(* CODESYS project IODev.library
   Company: ESO
   Description: Local Device Control - LDC IODevLibrary based on State Machine
   Version: 1.1.1.0
   Placeholder: ESO LDC IODev Library
   Author: Dan Popovic
   Title: ESO LDC IODev Library

Project tree, tasks and I/O mapping:
  libraries: Tc2_Standard, * (Beckhoff Automation GmbH); Tc2_System, * (Beckhoff Automation GmbH); Tc3_EventLogger, * (Beckhoff Automation GmbH); Tc3_Module, * (Beckhoff Automation GmbH); VisuSymbols, 3.5.10.0 (System)
  config/
    Device1_EtherCAT_SPLC014.xti
    Mappings_HW_SPLC014.xml
    Mappings_SIM.xml
  00000000-0000-0000-0000-000000000000|config\Device1_EtherCAT_SPLC014.xti
  00000000-0000-0000-0000-000000000000|config\Mappings_HW_SPLC014.xml
  00000000-0000-0000-0000-000000000000|config\Mappings_SIM.xml
  doc/
  DUTs/
    Enumerated/
      data type E_IODEV_COMMAND
      data type E_IODEV_CONVERSION
      data type E_IODEV_ERROR
      data type E_IODEV_EVENT
      data type E_IODEV_RPC_ERROR
      data type E_IODEV_STATE
      data type E_IODEV_STATUS
      data type E_IODEV_SUBSTATE
    Structures/
      data type T_IODEV_CFG
      data type T_IODEV_CTRL
      data type T_IODEV_INFO
      data type T_IODEV_STAT
  GVLs/
  lib/
  POUs/
    Channels/
      function block FB_IODEV_CH_ANALOG [ST]
      function block FB_IODEV_CH_ANLG_IN [ST]: M_Compute, M_Configure, M_Reset
      function block FB_IODEV_CH_ANLG_OUT [ST]: M_Compute, M_Configure, M_Reset
      function block FB_IODEV_CH_DIG_IN [ST]: M_Compute, M_Configure, M_Reset
      function block FB_IODEV_CH_DIG_OUT [ST]: M_Compute, M_Configure, M_Reset
      function block FB_IODEV_CH_DIGITAL [ST]
      function block FB_IODEV_CH_REAL [ST]
      function block FB_IODEV_CH_REAL_IN [ST]: M_Compute, M_Configure, M_Reset
      function block FB_IODEV_CHANNEL [ST]: M_Compute, M_Reset
    Examples/
      function block FB_IODEV_2_4_2_2_USER_CONFIG [ST]: M_UserConfigure
      function block FB_SENS_2_4A_2R_USER_CONFIG [ST]: M_UserConfigure
      function block FB_SENS_8_4 [ST]
      function block FB_SENS_8_4_USER_CONFIG [ST]: M_UserConfigure
      data type T_IODEV_CTRL_2_2
      data type T_IODEV_STAT_2_4
      data type T_IODEV_STAT_2_4A_2R
      data type T_IODEV_STAT_8_4
    Simulation/
      function block FB_SIM_SIGNAL_ANALOG [ST]
      function block FB_SIM_SIGNAL_DIGITAL [ST]
      function block FB_SIM_SIGNAL_REAL [ST]
    function block FB_IODEV_BASE [ST]: ActionDisableExecute, ActionEnableExecute, ActionErrExecute, ActionInitExecute, ActionResetExecute, ActionSetExecute, ActionStopExecute, ActionUnexpExecute, ActivityMonitoring, CheckForEvents, M_Configure, M_GetRpcErrorText, M_LogEventDebug, M_LogEventError, M_LogEventGeneral, M_ReadSensors, M_ResetConfig, M_ResetOutputs, M_SetOutputs, M_SetRpcStatus, M_UserConfigure, ProcessEvents, RPC_Disable, RPC_Enable, RPC_Init, RPC_Reset, RPC_SetDebug, RPC_SetLog, RPC_SetOutputs, RPC_Stop, SetAction, SetEvent, SetLastCommand, SetState, SetStatus
    program MAIN [ST]
  Version/
    global variables Global_Version
  VISUs/
    Templates/
      visualisation GUI_TEMPLATE_IODEV
    visualisation GUI_IODev001
    visualisation GUI_IODev002
  text list GlobalTextList
*)

// DUTs/Enumerated/E_IODEV_COMMAND
{attribute 'qualified_only'}
{attribute 'strict'}
TYPE E_IODEV_COMMAND :
(
	NONE	:= 0,
	
	RESET,
	INIT,
	STOP,
	ENABLE,
	DISABLE,
	SET_OUTPUTS
	
);
END_TYPE

// DUTs/Enumerated/E_IODEV_CONVERSION
TYPE E_IODEV_CONVERSION :
(
	CONVERSION_IODEV_NONE	:= 0,
	
	// Digital signals
	CONVERSION_IODEV_DIGITAL,
	// Analog signals
	CONVERSION_IODEV_LINEAR,
	CONVERSION_IODEV_QUADRATIC,
	CONVERSION_IODEV_EXP,
	CONVERSION_IODEV_EXP10
	
);
END_TYPE

// DUTs/Enumerated/E_IODEV_ERROR
{attribute 'qualified_only'}
{attribute 'strict'}
TYPE E_IODEV_ERROR :
(
	OK					:= 0,
	HW_NOT_OP			:= 1,			
	WRONG_CMD			:= 2,			
	INIT_FAILURE		:= 3,		

	NOT_INITIALISED		:= 90,
	ZERO_POINTER		:= 100	// Simulator error
);
END_TYPE

// DUTs/Enumerated/E_IODEV_EVENT
{attribute 'qualified_only'}
{attribute 'strict'}
TYPE E_IODEV_EVENT :
(
	NONE	:= 0,
	
	(* events corresponding to commands *)
	RESET,
	INIT,
	STOP,
	ENABLE,
	DISABLE,
	SET,
	
	(* 
		Events corresponding to internal events 
	*)
	INITDONE,
	
	
	(* events mapped to HW signals *)
	HWOK,
	ERRHW,
	ERRINIT
	
);
END_TYPE

// DUTs/Enumerated/E_IODEV_RPC_ERROR
{attribute 'qualified_only'}
{attribute 'strict'}
TYPE E_IODEV_RPC_ERROR :
(
	OK						:= 0,
	NOT_OP					:= -1,			
	NOT_NOTOP_READY			:= -2,			
	NOT_NOTOP_NOTREADY		:= -3,			
	LOCAL					:= -4			
);
END_TYPE

// DUTs/Enumerated/E_IODEV_STATE
{attribute 'qualified_only'}
{attribute 'strict'}
TYPE E_IODEV_STATE :
(
	NONE	:= 0,
	NOTOP,
	OP
);
END_TYPE

// DUTs/Enumerated/E_IODEV_STATUS
{attribute 'qualified_only'}
{attribute 'strict'}
TYPE E_IODEV_STATUS :
(
	OK		:= 0,
	ERROR
);
END_TYPE

// DUTs/Enumerated/E_IODEV_SUBSTATE
// Substates MUST match definitions in the WS driver that can be found in
// ICS/ifw/fcf/devmgr/devices/src/include/devmgr/devices/sensorConfig.hpp
// Never change them without consulting the Instrumentation SW team.
{attribute 'qualified_only'}
{attribute 'strict'}
TYPE E_IODEV_SUBSTATE :
(
	NONE			:= 0,
	
	NOTOP_NOTREADY	:= 100,
	NOTOP_READY		:= 101,
	NOTOP_ERROR		:= 199,
	
	OP_MONITORING	:= 200,
	OP_ERROR		:= 299
);
END_TYPE

// DUTs/Structures/T_IODEV_CFG
TYPE T_IODEV_CFG :
STRUCT
	sName:				STRING	:= 'IODev';	// Instance name
	bAutoOp:			BOOL 	:= FALSE;	// If TRUE, go automatically to OPERATIONAL state
	bUserConfig:		BOOL 	:= TRUE;	// If true, configuration in M_Configure() is used.
	
	nNum_DI:			INT		:= 0; 		// Number of digital INPUT signals
	nNum_AI:			INT		:= 0; 		// Number of analog INPUT signals of type INT
	nNum_RI:			INT		:= 0; 		// Number of analog INPUT signals of type REAL
	nNum_DisI:			INT		:= 0; 		// Number of discrete INPUT signals
	nNum_TI:			INT		:= 0; 		// Number of text INPUT signals
	
	nNum_DO:			INT		:= 0; 		// Number of digital OUTPUT signals
	nNum_AO:			INT		:= 0; 		// Number of analog OUTPUT signals of type INT
	nNum_DisO:			INT		:= 0; 		// Number of discrete OUTPUT signals
	nNum_TO:			INT		:= 0; 		// Number of text OUTPUT signals
	
	// Logging
	bLogExtTime:		BOOL 	:= FALSE;		// If TRUE, use external time in event logs. Default FALSE.
	bDebug:				BOOL 	:= FALSE;		// If TRUE, show event logs of Debug type. Default FALSE.
	bLog:				BOOL 	:= TRUE;		// If TRUE, log events. Default TRUE.
	
END_STRUCT
END_TYPE

// DUTs/Structures/T_IODEV_CTRL
TYPE T_IODEV_CTRL :
STRUCT
	nCommand:	E_IODEV_COMMAND	:= E_IODEV_COMMAND.NONE; (* See E_IODEV_COMMAND *)
	bExecute:	BOOL;
	
END_STRUCT
END_TYPE

// DUTs/Structures/T_IODEV_INFO
TYPE T_IODEV_INFO :
STRUCT
(*
Driver Information 

Change Log:
	0.1	2017-09-07	- First version - dummy implementation.
	0.2	2017-09-11	- Implemented digital/analog IN/OUT.
	0.3	2017-09-14	- Implemented digital/analog IN/OUT as FBs with methods.
					- Removed unused structures.
	0.6.0.0			- Restructure with pointers to channel arrays.
					- Removed input vars for number of channels. Defined in each derived FB.
					- Addition of FB_IODEV_SENS_8_4.
					- Addition of customised FB's.
	0.7.0.0			- Addition of stat.sLibVersion
	0.8.0.0			- RPC calls return INT.
					- Addition of E_IODEV_RPC_ERROR.
	0.8.0.1			- Addition of library category ESO/ELT.
	0.8.0.2			- Removed input parameters from OPC UA.
	0.9.0.0			- Renaming States STANDBY->NOTOP & FAILURE->ERROR.
	1.0.0.0			- WARNING: Requires TwinCAT 3.1 build 4022.20 or higher.
					- Projects need Tc3_EventLogger library included in References.
					- Addition of Methods for Event Logs.
					- Addition of cfg.bLog flag for enable/disable of logging.
					- Addition of RPC_SetDebug() and RPC_SetLog().
					- RPC calls not allowed in Local mode.
	1.0.0.1			- Compiled wit TwinCAT 3.1 build 4022.27.
					- Renamed TC_EVENTS.OpsEventClass to TC_EVENTS.IODevOpsEventClass.
					- Solved problem of 'growing' libraries by setting Property/Advanced/BuildAction to None for IODev.library and pdf files in dir config.
	1.0.0.2			- Pinned ST_IODevOpsEventClass under External Types.
	1.0.0.3			- Renumbered enumerations in E_IODEV_SUBSTATE to match WS.
	1.1.0.0			- Moved user defined structures under ctrl and stat.
					- Strict enumerated types.
					- Used RefCtrl and RefStat in BASE FB.
*)
	sDate:			STRING(32)	:= '2019-04-24';
	sDescription:	STRING(80) 	:= 'State Machine based IODev controller';
	sName:			STRING(64)	:= 'FB_IODEV';
	sPlatform:		STRING(32)	:= 'CoDeSys';
	sSynopsis:		STRING(64)	:= 'State Machine based IODev controller';
	nVersionMajor:	DINT		:= 1;
	nVersionMinor:	DINT		:= 1;
END_STRUCT
END_TYPE

// DUTs/Structures/T_IODEV_STAT
TYPE T_IODEV_STAT :
STRUCT
	bLocal:			BOOL	:= FALSE;						(* Device operated from PLC GUI *)

	nState:			E_IODEV_STATE	:= E_IODEV_STATE.NOTOP;				// State
	nSubstate:		E_IODEV_SUBSTATE:= E_IODEV_SUBSTATE.NOTOP_NOTREADY;	// Substate

	nErrorCode: 	E_IODEV_ERROR 	:= E_IODEV_ERROR.OK;		(* Error code *)
	nLastCommand:	E_IODEV_COMMAND	:= E_IODEV_COMMAND.NONE;	(* Last command sent to the device *)
	nRpcErrorCode: 	E_IODEV_RPC_ERROR 	:= E_IODEV_RPC_ERROR.OK;(* RPC Error code *)
	nStatus: 		E_IODEV_STATUS	:= E_IODEV_STATUS.OK; 		(* Device status *)

	sState:			STRING	:= 'NOT OP';					(* State textual description *)
	sSubstate:		STRING	:= 'NOT READY';					(* Substate textual description *)
	sErrorText: 	STRING 	:= 'OK'; 						(* Error text *)
	sRPCErrorText: 	STRING 	:= 'OK'; 						(* RPC Error text *)
	sStatus: 		STRING 	:= 'OK'; 						(* Status in textual form, e.g. 'OFF' *)
	sLastCommand:	STRING	:= 'NONE';						(* Last command, as string, sent to the device *)
	sLibVersion:	STRING	:= 'UNKNOWN';					(* Library version as string, e.g. '1.2.0.0' *)
	
	sActionDesc:	STRING	:= '';
	sEventDesc:		STRING	:= '';

	nCycleCounter:	UDINT	:= 0;	// Alive flag
END_STRUCT
END_TYPE

// POUs/Examples/T_IODEV_CTRL_2_2
// EXAMPLE:	Extension of T_IODEV_CTRL with 2 DO and 2 AO.
// 			Used in FB_IODEV_2_4_2_2_USER_CONFIG.
TYPE T_IODEV_CTRL_2_2 EXTENDS T_IODEV_CTRL :
STRUCT
	// Signals, Outputs
	arrDO:	ARRAY [0..1] OF FB_IODEV_CH_DIG_OUT;	// 2 digital outputs
	arrAO:	ARRAY [0..1] OF FB_IODEV_CH_ANLG_OUT;	// 2 analog outputs
END_STRUCT
END_TYPE

// POUs/Examples/T_IODEV_STAT_2_4
// EXAMPLE:	Extension of T_IODEV_STAT with 2 DI and 4 AI.
// 			Used in FB_IODEV_2_4_2_2_USER_CONFIG.
TYPE T_IODEV_STAT_2_4 EXTENDS T_IODEV_STAT :
STRUCT
	//
	// Signals, inputs.
	//
	arrDI:	ARRAY [0..1] OF FB_IODEV_CH_DIG_IN;		// 2 digital inputs
	arrAI:	ARRAY [0..3] OF FB_IODEV_CH_ANLG_IN;	// 4 analog inputs
END_STRUCT
END_TYPE

// POUs/Examples/T_IODEV_STAT_2_4A_2R
// EXAMPLE:	Extension of T_IODEV_STAT with 2 DI and 4 AI of type INT and 2 AI of type REAL.
// 			Used in FB_SENS_2_4A_2R_USER_CONFIG.
TYPE T_IODEV_STAT_2_4A_2R EXTENDS T_IODEV_STAT :
STRUCT
	//
	// Signals, inputs.
	//
	arrDI:	ARRAY [0..1] OF FB_IODEV_CH_DIG_IN;		// 2 digital inputs
	arrAI:	ARRAY [0..3] OF FB_IODEV_CH_ANLG_IN;	// 4 analog inputs of type INT
	arrRI:	ARRAY [0..1] OF FB_IODEV_CH_REAL_IN;	// 2 analog inputs of type REAL
END_STRUCT
END_TYPE

// POUs/Examples/T_IODEV_STAT_8_4
// EXAMPLE:	Extension of T_IODEV_STAT with 8 DI and 4 AI.
// 			Used in FB_SENS_8_4.
TYPE T_IODEV_STAT_8_4 EXTENDS T_IODEV_STAT :
STRUCT
	//
	// Signals, inputs.
	//
	arrDI:	ARRAY [0..7] OF FB_IODEV_CH_DIG_IN;		// 8 digital inputs
	arrAI:	ARRAY [0..3] OF FB_IODEV_CH_ANLG_IN;	// 4 analog inputs
END_STRUCT
END_TYPE

// Version/Global_Version
{attribute 'TcGenerated'}
{attribute 'no-analysis'}
{attribute 'linkalways'}
// This function has been automatically generated from the project information.
VAR_GLOBAL CONSTANT
	{attribute 'const_non_replaced'}
	stLibVersion_ESO_LDC_IODev_Library : ST_LibVersion := (iMajor := 1, iMinor := 1, iBuild := 1, iRevision := 0, nFlags := 0, sVersion := '1.1.1.0');
END_VAR

// POUs/Channels/FB_IODEV_CH_ANALOG
FUNCTION_BLOCK FB_IODEV_CH_ANALOG EXTENDS FB_IODEV_CHANNEL
VAR_INPUT
END_VAR
VAR_OUTPUT
END_VAR
VAR
	// Configuration parameters
	// Configured for R/W OPC UA Data Access !!!
	{attribute 'OPC.UA.DA' := '1'}
	{attribute 'OPC.UA.DA.Access' := '3'}
	nConversion:	E_IODEV_CONVERSION	:= CONVERSION_IODEV_NONE;
	{attribute 'OPC.UA.DA' := '1'}
	{attribute 'OPC.UA.DA.Access' := '3'}
	lrPar1:			LREAL 	:= 0.0;
	{attribute 'OPC.UA.DA' := '1'}
	{attribute 'OPC.UA.DA.Access' := '3'}
	lrPar2:			LREAL 	:= 0.0;
	{attribute 'OPC.UA.DA' := '1'}
	{attribute 'OPC.UA.DA.Access' := '3'}
	lrPar3:			LREAL 	:= 0.0;

END_VAR

END_FUNCTION_BLOCK

// POUs/Channels/FB_IODEV_CHANNEL
FUNCTION_BLOCK FB_IODEV_CHANNEL
VAR_INPUT
END_VAR
VAR_OUTPUT
END_VAR
VAR
END_VAR

METHOD M_Compute
VAR_INPUT
END_VAR
END_METHOD

METHOD M_Reset
VAR_INPUT
END_VAR
END_METHOD

END_FUNCTION_BLOCK

// POUs/Channels/FB_IODEV_CH_ANLG_IN
FUNCTION_BLOCK FB_IODEV_CH_ANLG_IN EXTENDS FB_IODEV_CH_ANALOG
VAR_INPUT
END_VAR
VAR_OUTPUT
END_VAR
VAR
	// Physical input signal
	// No access via OPC UA.
	{attribute 'OPC.UA.DA' := '0'}
	i_nValue	AT %I*:	INT;

	// Status - OPC UA Read only
	{attribute 'OPC.UA.DA' := '1'}
	{attribute 'OPC.UA.DA.Access' := '1'}
	nValue:			INT;	// Raw input value
	{attribute 'OPC.UA.DA' := '1'}
	{attribute 'OPC.UA.DA.Access' := '1'}
	lrValueUser:	LREAL;	// Computed value in User Units
	
END_VAR

METHOD M_Compute
VAR_INPUT
END_VAR
VAR
	lrValue:	LREAL;
END_VAR
nValue	:= i_nValue;
lrValue	:= INT_TO_LREAL(i_nValue);

CASE nConversion OF
	CONVERSION_IODEV_NONE:
		lrValueUser	:= lrValue;
	CONVERSION_IODEV_LINEAR:
		lrValueUser	:= lrPar1 * lrValue  +  lrPar2;
	CONVERSION_IODEV_QUADRATIC:
		lrValueUser	:= lrPar1 * lrValue * lrValue  +  lrPar2 * lrValue  +  lrPar3;
	CONVERSION_IODEV_EXP:
		lrValueUser	:= EXP (lrPar1 * lrValue  +  lrPar2);
	CONVERSION_IODEV_EXP10:
		lrValueUser	:= EXPT (10.0, (lrPar1 * lrValue  +  lrPar2));
END_CASE
END_METHOD

METHOD M_Configure
VAR_INPUT
END_VAR
VAR_INPUT
	in_eConversion:	E_IODEV_CONVERSION;
	in_lrPar1:		LREAL := 0.0;
	in_lrPar2:		LREAL := 0.0;
	in_lrPar3:		LREAL := 0.0;
END_VAR
nConversion		:= in_eConversion;
lrPar1			:= in_lrPar1;
lrPar2			:= in_lrPar2;
lrPar3			:= in_lrPar3;
END_METHOD

METHOD M_Reset
VAR_INPUT
END_VAR
nConversion	:= CONVERSION_IODEV_NONE;
lrPar1			:= 0.0;
lrPar2			:= 0.0;
lrPar3			:= 0.0;

nValue			:= 0;
lrValueUser		:= 0.0;
END_METHOD

END_FUNCTION_BLOCK

// POUs/Channels/FB_IODEV_CH_ANLG_OUT
FUNCTION_BLOCK FB_IODEV_CH_ANLG_OUT EXTENDS FB_IODEV_CH_ANALOG
VAR_INPUT
END_VAR
VAR_OUTPUT
END_VAR
VAR
	// Physical output signal
	// No access via OPC UA.
	{attribute 'OPC.UA.DA' := '0'}
	q_nValue	AT %Q*:	INT;

	// Output values
	// Configured for R/W OPC UA Data Access !!!
	{attribute 'OPC.UA.DA' := '1'}
	{attribute 'OPC.UA.DA.Access' := '3'}
	nValue:			INT;	// Computed output value
	{attribute 'OPC.UA.DA' := '1'}
	{attribute 'OPC.UA.DA.Access' := '3'}
	lrValueUser:	LREAL;	// Output value in User Units
	
END_VAR

METHOD M_Compute
VAR_INPUT
END_VAR
//
// For CONVERSION_IODEV_NONE nValue is used for output.
// In this case nValue is copied into lrValueUser.
// For others nValue is calculated from the User value.
//
CASE nConversion OF
	CONVERSION_IODEV_NONE:
		lrValueUser := INT_TO_LREAL(nValue);	// Copy nValue into lrValueUser
	CONVERSION_IODEV_LINEAR:
		nValue	:= LREAL_TO_INT(lrPar1 * lrValueUser  +  lrPar2);
	CONVERSION_IODEV_QUADRATIC:
		nValue	:= LREAL_TO_INT(lrPar1 * lrValueUser * lrValueUser  +  lrPar2 * lrValueUser  +  lrPar3);
	CONVERSION_IODEV_EXP:
		nValue	:= LREAL_TO_INT(EXP (lrPar1 * lrValueUser  +  lrPar2));
	CONVERSION_IODEV_EXP10:
		nValue	:= LREAL_TO_INT(EXPT (10.0, (lrPar1 * lrValueUser  +  lrPar2)));
END_CASE

// Set the output
q_nValue	:= nValue;
END_METHOD

METHOD M_Configure
VAR_INPUT
END_VAR
VAR_INPUT
	in_eConversion:	E_IODEV_CONVERSION;
	in_lrPar1:		LREAL := 0.0;
	in_lrPar2:		LREAL := 0.0;
	in_lrPar3:		LREAL := 0.0;
END_VAR
nConversion		:= in_eConversion;
lrPar1			:= in_lrPar1;
lrPar2			:= in_lrPar2;
lrPar3			:= in_lrPar3;

// Set output to zero
q_nValue		:= 0;
nValue			:= 0;
lrValueUser		:= 0.0;
END_METHOD

METHOD M_Reset
VAR_INPUT
END_VAR
nConversion	:= CONVERSION_IODEV_NONE;
lrPar1			:= 0.0;
lrPar2			:= 0.0;
lrPar3			:= 0.0;

// Set output to zero
q_nValue		:= 0;
nValue			:= 0;
lrValueUser		:= 0.0;
END_METHOD

END_FUNCTION_BLOCK

// POUs/Channels/FB_IODEV_CH_DIG_IN
FUNCTION_BLOCK FB_IODEV_CH_DIG_IN EXTENDS FB_IODEV_CH_DIGITAL
VAR_INPUT
END_VAR
VAR_OUTPUT
END_VAR
VAR
	// Physical input signal.
	// No access via OPC UA.
	{attribute 'OPC.UA.DA' := '0'}
	i_bValue	AT %I*:	BOOL;

	// Status - OPC UA Read only
	{attribute 'OPC.UA.DA' := '1'}
	{attribute 'OPC.UA.DA.Access' := '1'}
	bValue:		BOOL;
	{attribute 'OPC.UA.DA' := '1'}
	{attribute 'OPC.UA.DA.Access' := '1'}
	sValueUser:	STRING(16)	:= '0';

END_VAR

// Nothing to do
;

METHOD M_Compute
VAR_INPUT
END_VAR
// Read Digital INPUT and update labels
bValue	:= i_bValue;

IF bValue THEN
	sValueUser	:= sLabel_1;
ELSE
	sValueUser	:= sLabel_0;
END_IF
END_METHOD

METHOD M_Configure
VAR_INPUT
	in_sLabel_0:	STRING(16)	:= '0';
	in_sLabel_1:	STRING(16)	:= '1';
END_VAR
// Set labels
sLabel_0	:= in_sLabel_0;
sLabel_1	:= in_sLabel_1;
END_METHOD

METHOD M_Reset
VAR_INPUT
END_VAR
sLabel_0	:= '0';
sLabel_1	:= '1';

bValue		:= FALSE;
sValueUser	:= sLabel_0;
END_METHOD

END_FUNCTION_BLOCK

// POUs/Channels/FB_IODEV_CH_DIGITAL
FUNCTION_BLOCK FB_IODEV_CH_DIGITAL EXTENDS FB_IODEV_CHANNEL
VAR_INPUT
END_VAR
VAR_OUTPUT
END_VAR
VAR
	// Configuration parameters
	// Configured for R/W OPC UA Data Access !!!
	{attribute 'OPC.UA.DA' := '1'}
	{attribute 'OPC.UA.DA.Access' := '3'}
	sLabel_0:	STRING(16)	:= '0';
	{attribute 'OPC.UA.DA' := '1'}
	{attribute 'OPC.UA.DA.Access' := '3'}
	sLabel_1:	STRING(16)	:= '1';
END_VAR

END_FUNCTION_BLOCK

// POUs/Channels/FB_IODEV_CH_DIG_OUT
FUNCTION_BLOCK FB_IODEV_CH_DIG_OUT EXTENDS FB_IODEV_CH_DIGITAL
VAR_INPUT
END_VAR
VAR_OUTPUT
END_VAR
VAR
	// Physical output signal.
	// No access via OPC UA.
	{attribute 'OPC.UA.DA' := '0'}
	q_bValue	AT %Q*:	BOOL;

	// Set values 
	// Configured for R/W OPC UA Data Access !!!
	{attribute 'OPC.UA.DA' := '1'}
	{attribute 'OPC.UA.DA.Access' := '3'}
	bValue:		BOOL;
	{attribute 'OPC.UA.DA' := '1'}
	{attribute 'OPC.UA.DA.Access' := '3'}
	sValueUser:	STRING(16);
	
	// Configuration parameters
	// Configured for R/W OPC UA Data Access !!!
	{attribute 'OPC.UA.DA' := '1'}
	{attribute 'OPC.UA.DA.Access' := '3'}
	nConversion:	E_IODEV_CONVERSION	:= CONVERSION_IODEV_NONE;
END_VAR

METHOD M_Compute
VAR_INPUT
END_VAR
// Check if the digital output should be calculated from User labels.
// If yes, convert user label to digital output value.
// Otherwise, just take the value from bValue and set the labels.
IF nConversion = CONVERSION_IODEV_DIGITAL THEN
	IF sValueUser = sLabel_0 THEN
		bValue	:= FALSE;
	ELSIF sValueUser = sLabel_1 THEN
		bValue	:= TRUE;
	END_IF
ELSE
	IF bValue THEN
		sValueUser	:= sLabel_1;
	ELSE
		sValueUser	:= sLabel_0;
	END_IF
END_IF

// Set output
q_bValue	:= bValue;
END_METHOD

METHOD M_Configure
VAR_INPUT
	in_nConversion:	INT			:= CONVERSION_IODEV_NONE;	// CONVERSION_IODEV_NONE or CONVERSION_IODEV_DIGITAL
	in_sLabel_0:	STRING(16)	:= '0';
	in_sLabel_1:	STRING(16)	:= '1';
END_VAR
// Set conversion type
nConversion	:= in_nConversion;

// Set labels
sLabel_0	:= in_sLabel_0;
sLabel_1	:= in_sLabel_1;

// Set output to zero
q_bValue	:= FALSE;
bValue		:= FALSE;
sValueUser	:= sLabel_0;
END_METHOD

METHOD M_Reset
VAR_INPUT
END_VAR
nConversion	:= CONVERSION_IODEV_NONE;
sLabel_0	:= '0';
sLabel_1	:= '1';

// Set output to zero
q_bValue	:= FALSE;
bValue		:= FALSE;
sValueUser	:= sLabel_0;
END_METHOD

END_FUNCTION_BLOCK

// POUs/Channels/FB_IODEV_CH_REAL
// FB for analog input signals of type REAL.
// The EL3692 is one of input terminals that provide inputs as REAL.
FUNCTION_BLOCK FB_IODEV_CH_REAL EXTENDS FB_IODEV_CHANNEL
VAR_INPUT
END_VAR
VAR_OUTPUT
END_VAR
VAR
	// Configuration parameters
	// Configured for R/W OPC UA Data Access !!!
	{attribute 'OPC.UA.DA' := '1'}
	{attribute 'OPC.UA.DA.Access' := '3'}
	nConversion:	E_IODEV_CONVERSION	:= CONVERSION_IODEV_NONE;
	{attribute 'OPC.UA.DA' := '1'}
	{attribute 'OPC.UA.DA.Access' := '3'}
	lrPar1:			LREAL 	:= 0.0;
	{attribute 'OPC.UA.DA' := '1'}
	{attribute 'OPC.UA.DA.Access' := '3'}
	lrPar2:			LREAL 	:= 0.0;
	{attribute 'OPC.UA.DA' := '1'}
	{attribute 'OPC.UA.DA.Access' := '3'}
	lrPar3:			LREAL 	:= 0.0;

END_VAR

END_FUNCTION_BLOCK

// POUs/Channels/FB_IODEV_CH_REAL_IN
FUNCTION_BLOCK FB_IODEV_CH_REAL_IN EXTENDS FB_IODEV_CH_REAL
VAR_INPUT
END_VAR
VAR_OUTPUT
END_VAR
VAR
	// Physical input signal
	// No access via OPC UA.
	{attribute 'OPC.UA.DA' := '0'}
	i_rValue	AT %I*:	REAL;	// Physical input signal as REAL

	// Status - OPC UA Read only
	{attribute 'OPC.UA.DA' := '1'}
	{attribute 'OPC.UA.DA.Access' := '1'}
	lrValue:		LREAL;	// Raw input value converted from REAL (float) to LREAL (double)
	{attribute 'OPC.UA.DA' := '1'}
	{attribute 'OPC.UA.DA.Access' := '1'}
	lrValueUser:	LREAL;	// Computed value from lrValue in User Units
	
END_VAR

METHOD M_Compute
VAR_INPUT
END_VAR
VAR
END_VAR
lrValue	:= REAL_TO_LREAL(i_rValue);

CASE nConversion OF
	CONVERSION_IODEV_NONE:
		lrValueUser	:= lrValue;
	CONVERSION_IODEV_LINEAR:
		lrValueUser	:= lrPar1 * lrValue  +  lrPar2;
	CONVERSION_IODEV_QUADRATIC:
		lrValueUser	:= lrPar1 * lrValue * lrValue  +  lrPar2 * lrValue  +  lrPar3;
	CONVERSION_IODEV_EXP:
		lrValueUser	:= EXP (lrPar1 * lrValue  +  lrPar2);
	CONVERSION_IODEV_EXP10:
		lrValueUser	:= EXPT (10.0, (lrPar1 * lrValue  +  lrPar2));
END_CASE
END_METHOD

METHOD M_Configure
VAR_INPUT
END_VAR
VAR_INPUT
	in_eConversion:	E_IODEV_CONVERSION;
	in_lrPar1:		LREAL := 0.0;
	in_lrPar2:		LREAL := 0.0;
	in_lrPar3:		LREAL := 0.0;
END_VAR
nConversion		:= in_eConversion;
lrPar1			:= in_lrPar1;
lrPar2			:= in_lrPar2;
lrPar3			:= in_lrPar3;
END_METHOD

METHOD M_Reset
VAR_INPUT
END_VAR
nConversion	:= CONVERSION_IODEV_NONE;
lrPar1			:= 0.0;
lrPar2			:= 0.0;
lrPar3			:= 0.0;

lrValue			:= 0.0;
lrValueUser		:= 0.0;
END_METHOD

END_FUNCTION_BLOCK

// POUs/Examples/FB_IODEV_2_4_2_2_USER_CONFIG
// EXAMPLE: Customised FB_IODEV_BASE for 2 DI, 4 AI, 2 DO and 2 AO.
//          Overloaded M_UserConfigure() method for User Configuration of channels.
FUNCTION_BLOCK FB_IODEV_2_4_2_2_USER_CONFIG EXTENDS FB_IODEV_BASE
VAR_INPUT
END_VAR
VAR_OUTPUT
END_VAR
VAR
	// Control parameters that EXTEND T_IODEV_CTRL
	{attribute 'OPC.UA.DA' := '1'}
	ctrl:	T_IODEV_CTRL_2_2;	
	// Status parameters that EXTEND T_IODEV_STAT
	{attribute 'OPC.UA.DA' := '1'}
	{attribute 'OPC.UA.DA.Access' := '1'}
	stat:	T_IODEV_STAT_2_4;	
END_VAR

//
// TODO_USER
//
//
// Set References
RefCtrl	REF=ctrl;
RefStat	REF=stat;

// Set number of channels for each type.
// Default values are set to zero.
// Set whatever is not zero, i.e. whatever is defined.
// WARNING: The values MUST match the sizes of corresponding arrays above !!!
//
cfg.nNum_DI		:=	2; 	// Number of digital INPUT signals, arrDI:	ARRAY [0..1]
cfg.nNum_AI		:=	4; 	// Number of analog INPUT signals,  arrAI:	ARRAY [0..3]
//cfg.nNum_DisI	:=	0; 	// Number of discrete INPUT signals
//cfg.nNum_TI	:=	0; 	// Number of text INPUT signals

cfg.nNum_DO		:=	2; 	// Number of digital OUTPUT signals, arrDO:	ARRAY [0..1]
cfg.nNum_AO		:=	2; 	// Number of analog OUTPUT signals,  arrAO:	ARRAY [0..1]
//cfg.nNum_DisO	:=	0; 	// Number of discrete OUTPUT signals
//cfg.nNum_TO	:=	0; 	// Number of text OUTPUT signals

//
// Set pointers for EXISTING arrays ONLY, e.g. arrDI, arrAI, etc.
//
pArrDI	:= ADR(stat.arrDI[0]);
pArrAI	:= ADR(stat.arrAI[0]);
pArrDO	:= ADR(ctrl.arrDO[0]);
pArrAO	:= ADR(ctrl.arrAO[0]);

//
// Execute the base class object FB_IODEV_BASE
//
SUPER^();

// TODO_USER
//
// Define individual channel configurations, if used.
METHOD M_UserConfigure
VAR_INPUT
END_VAR
// TODO_USER
//
// Example implementation.
// Hard code any signal configuration.
//

// Configuration parameter cfg.bUserConfig defines if 
// the hard-coded configuration below should be used or
// the signals will be configured from the WS.

//
// Digital signals
//
// Digital inputs (defined in stat structure T_IODEV_STAT_CUSTOM)
// Signal DI[0] is a door open signal
// Signal DI[1] is a light switch signal
stat.arrDI[0].M_Configure('CLOSED', 'OPEN');
stat.arrDI[1].M_Configure('OFF',    'ON');

// Digital outputs (defined in ctrl structure T_IODEV_CTRL_CUSTOM)
// Signal DO[0] is a pure digital signal without user defined labels
// Signal DO[1] is a light switch signal that is controlled by setting User labels 'OFF' and 'ON'.
ctrl.arrDO[0].M_Configure(CONVERSION_IODEV_NONE, 	'0', 	'1');
ctrl.arrDO[1].M_Configure(CONVERSION_IODEV_DIGITAL,	'OFF',	'ON');


//
// Analog signals
//
// Analog inputs (defined in stat structure T_IODEV_STAT_CUSTOM)
stat.arrAI[0].M_Configure(CONVERSION_IODEV_NONE, 		0.0,   0.0, 0.0);
stat.arrAI[1].M_Configure(CONVERSION_IODEV_LINEAR, 		2.0,   1.0, 0.0);
stat.arrAI[2].M_Configure(CONVERSION_IODEV_QUADRATIC,	2.0,   1.0, 5.0);
// Edwards pressure guage
// P =10^(1.5*V - 12)    [mbar]
// 16-bit A/D converter, +=10V, e.g. EL3102.
// 1V = 2^16/10/2 = 3276.8 bit
// P = 10^(1.5*V - 12) = 10^(1.5/3276.8*bit - 12) = 10^(0.000457763*bit - 12)
stat.arrAI[3].M_Configure(CONVERSION_IODEV_EXP10, 	0.000457763, -12.0, 0.0);	

//
// Analog outputs (defined in ctrl structure T_IODEV_CTRL_CUSTOM)
ctrl.arrAO[0].M_Configure(CONVERSION_IODEV_NONE, 	0.0,   0.0, 0.0);	// No conversion
ctrl.arrAO[1].M_Configure(CONVERSION_IODEV_LINEAR, 	0.1,   0.0, 0.0);	// out = User/10
END_METHOD

END_FUNCTION_BLOCK

// POUs/FB_IODEV_BASE
FUNCTION_BLOCK FB_IODEV_BASE
VAR_INPUT
	{attribute 'OPC.UA.DA':='0'}
	in_sName:		STRING	:= 'IODev';	// Instance name
	{attribute 'OPC.UA.DA':='0'}
	in_bAutoOp:		BOOL 	:= FALSE;	// If TRUE, go automatically to OPERATIONAL state. Default FALSE.
	{attribute 'OPC.UA.DA':='0'}
	in_bUserConfig:	BOOL 	:= FALSE;	// If TRUE, configuration in M_UserConfigure() is used. Default FALSE.
END_VAR
VAR_OUTPUT
END_VAR
VAR RETAIN
END_VAR
VAR
	{attribute 'OPC.UA.DA' := '1'}
	cfg:		T_IODEV_CFG;	
	{attribute 'OPC.UA.DA' := '0'}
	RefCtrl:	REFERENCE TO T_IODEV_CTRL;	
	{attribute 'OPC.UA.DA' := '1'}
	{attribute 'OPC.UA.DA.Access' := '1'}
	info:		T_IODEV_INFO;	(* ReadOnly *)
	{attribute 'OPC.UA.DA' := '0'}
	RefStat:	REFERENCE TO T_IODEV_STAT;	    // Reference to Status parameters

	{attribute 'OPC.UA.DA' := '0'}
	nEvent:		      	DINT := E_IODEV_EVENT.NONE;
	{attribute 'OPC.UA.DA' := '0'}
	nInternalEvent:		DINT := E_IODEV_EVENT.NONE;
	
	// Pointers to I/O data to be defined in FB's that inherit from this BASE FB.
	// In the BASE FB they are set to zero to prevent any access to data.
	pArrDI:	POINTER TO FB_IODEV_CH_DIG_IN	:= 0;	// pointer to DI
	pArrAI:	POINTER TO FB_IODEV_CH_ANLG_IN	:= 0;	// pointer to AI
	pArrRI:	POINTER TO FB_IODEV_CH_REAL_IN	:= 0;	// pointer to RI
	pArrDO:	POINTER TO FB_IODEV_CH_DIG_OUT	:= 0;	// pointer to DO
	pArrAO:	POINTER TO FB_IODEV_CH_ANLG_OUT	:= 0;	// pointer to AO

	
	// Operational Events
	{attribute 'OPC.UA.DA' := '0'}
	fbEventError:	FB_TcMessage;
	{attribute 'OPC.UA.DA' := '0'}
	fbEventDebug:	FB_TcMessage;
	{attribute 'OPC.UA.DA' := '0'}
	fbEventGeneral:	FB_TcMessage;
	
	(***** Physical signals - to be mapped!!! *****)

	(* Outputs *)

	(* Inputs *)	
	{attribute 'OPC.UA.DA' := '0'}
	i_nCouplerState	AT %I*: 	UINT;	(* Link it to Coupler->InfoData->State *)

	// Flag if the device is ready to receive commands.
	// It takes a couple of cycles for the system to read inputs after reboot.
	{attribute 'OPC.UA.DA' := '0'}
	bDeviceNotReady:		BOOL 	:= TRUE;
	

END_VAR

// On first cycle configure from input params and internally execute M_UserConfigure()
IF bDeviceNotReady THEN
	// Set device Configuration
	M_Configure();
	RETURN;
END_IF

// Increment counter.
// This will be seen as 'alive' flag.
RefStat.nCycleCounter	:= RefStat.nCycleCounter + 1;


(* === Check for commands and internal events to be processed === *)
CheckForEvents();

(* === Process events according to the State Machine === *)
ProcessEvents();

METHOD ActionDisableExecute
VAR_INPUT
END_VAR
SetAction('ActionDisableExecute');

// Log event
M_LogEventGeneral('DISABLE executed.');

// Reset all outputs
M_ResetOutputs();
END_METHOD

METHOD ActionEnableExecute
VAR_INPUT
END_VAR
END_METHOD

METHOD ActionErrExecute
VAR_INPUT
END_VAR
SetAction('ActionErrExecute');

IF nEvent = E_IODEV_EVENT.ERRHW THEN
	SetStatus(E_IODEV_ERROR.HW_NOT_OP, 'ERROR: HW not in OP state');	
ELSIF nEvent = E_IODEV_EVENT.ERRINIT THEN
	SetStatus(E_IODEV_ERROR.INIT_FAILURE, 'ERROR: INIT failed');	
END_IF
END_METHOD

METHOD ActionInitExecute
VAR_INPUT
END_VAR
SetAction('ActionInitExecute');

// Apply User configuration if configured so
IF cfg.bUserConfig THEN
	M_UserConfigure();
END_IF

// Log event
M_LogEventGeneral('INIT executed.');


// Clear any error
SetStatus(E_IODEV_ERROR.OK, 'OK');

// Set INITDONE event
nInternalEvent 		:= E_IODEV_EVENT.INITDONE;
END_METHOD

METHOD ActionResetExecute
VAR_INPUT
END_VAR
SetAction('ActionResetExecute');

M_ResetConfig();	// Reset existing User configuration

// Log event
M_LogEventGeneral('RESET executed.');


// Clear any error
SetStatus(E_IODEV_ERROR.OK, 'OK');
END_METHOD

METHOD ActionSetExecute
VAR_INPUT
END_VAR
SetAction('ActionSetExecute');

// Log event
M_LogEventGeneral('SET executed. Outputs activated.');

(* Clear the error *)
SetStatus(E_IODEV_ERROR.OK,'OK');

// Set Outputs
M_SetOutputs();
END_METHOD

METHOD ActionStopExecute
VAR_INPUT
END_VAR
SetAction('ActionStopExecute');

// Reset all outputs
M_ResetOutputs();
END_METHOD

METHOD ActionUnexpExecute
VAR_INPUT
END_VAR
SetAction('ActionUnexpExecute');

(*
	We don't want to overwrite initial error.
	Update error only if it is currently equal to OK. 
*)
IF RefStat.nErrorCode = E_IODEV_ERROR.OK THEN
	IF nEvent = E_IODEV_EVENT.ERRHW THEN
		RefStat.nErrorCode		:= E_IODEV_ERROR.HW_NOT_OP;
		RefStat.sErrorText		:= 'ERROR: HW not in OP state.';	
	ELSIF nEvent = E_IODEV_EVENT.ERRINIT THEN
		RefStat.nErrorCode		:= E_IODEV_ERROR.INIT_FAILURE;
		RefStat.sErrorText		:= 'ERROR: INIT failed.';	
	END_IF
END_IF
END_METHOD

METHOD ActivityMonitoring
VAR_INPUT
END_VAR
SetAction('ActivityMonitoring');

IF	i_nCouplerState <> 8  THEN
	nInternalEvent 		:= E_IODEV_EVENT.ERRHW;

	SetStatus(E_IODEV_ERROR.HW_NOT_OP, 'HW not in OP state');	
	RETURN;
END_IF

// Read all sensors define in the system
M_ReadSensors();
END_METHOD

METHOD CheckForEvents
VAR_INPUT
END_VAR

(* 
	Start assuming the HW is OK. 
	This is needed to recover from the situation where 
	the HW was failing and now it is working.
*)
nEvent := E_IODEV_EVENT.HWOK;




(* 
	Check for events in the following order: 
   	1) HW failure: without HW avilability there is no point to do anything
	2) Internal events: to allow completing the initiated commands before 
                        starting processing new commands. 
   	3) Commands: to react to external commands. Commands should be executed 
                 before processing HW signals to allow to start a recovery action.
   	4) HW signals: if any.
*)

IF i_nCouplerState <> 8 THEN	
	(* Check if the HW is NOT OK *)
	(*
	If the hardware status is NOT OK, we cannot trust the readings.
	Variable i_nCouplerState has to be mapped to a State of a terminal, e.g. EK1100.
	The value should be 8.
 	*)
	SetEvent(E_IODEV_EVENT.ERRHW);
	SetStatus(E_IODEV_ERROR.HW_NOT_OP, 'ERROR: HW not in OPERATIONAL state');

ELSIF nInternalEvent <> E_IODEV_EVENT.NONE THEN
	(* Handle internal events *)
	SetEvent(nInternalEvent);
	nInternalEvent := E_IODEV_EVENT.NONE;
ELSIF RefCtrl.bExecute = TRUE  THEN
	(* Handle commands *)
	RefCtrl.bExecute		:= FALSE;			(* Clear the Execute bit *)
	SetLastCommand(RefCtrl.nCommand);			(* Save the last command *)
	SetEvent(RefCtrl.nCommand);
	RefCtrl.nCommand 		:= E_IODEV_COMMAND.NONE;	(* Clear the Command *)
ELSE
	(* Handle HW problems and unexpected bahaviour *)
	
END_IF
END_METHOD

METHOD M_Configure : BOOL
VAR_INPUT
END_VAR
// If first cycle, copy configuration AND RETURN in order for the system to read all inputs before doing any work
IF RefStat.nCycleCounter = 0 THEN
	// Copy input parameters into configuration
	cfg.sName		:=	in_sName;		// Instance name

	cfg.bAutoOp		:=	in_bAutoOp;		// If TRUE, go automatically to OPERATIONAL state
	cfg.bUserConfig	:=	in_bUserConfig;	// If TRUE, configuration in M_UserConfigure() is used.
	
	// Get the version number 
	RefStat.sLibVersion	:= stLibVersion_ESO_LDC_IODev_Library.sVersion;

	// Increment counter.
	RefStat.nCycleCounter	:= RefStat.nCycleCounter + 1;
	RETURN;
ELSIF RefStat.nCycleCounter < 100 THEN
	// Give the system a couple of cycles
	// Increment counter.
	RefStat.nCycleCounter	:= RefStat.nCycleCounter + 1;
	RETURN;
END_IF

// After 100 cycles the system is read, e.g. coupler state is 8.

// Create Event instances
fbEventError.CreateEx	(TC_EVENTS.IODevOpsEventClass.Error,0);
fbEventDebug.CreateEx	(TC_EVENTS.IODevOpsEventClass.Debug,0);
fbEventGeneral.CreateEx	(TC_EVENTS.IODevOpsEventClass.General,0);


// The device is ready now.
bDeviceNotReady := FALSE;


// Clear errors
RefStat.nErrorCode		:= E_IODEV_ERROR.OK;
RefStat.sErrorText		:= 'OK';	


//
// Execute User configuration, if configured to do so.
//
IF cfg.bUserConfig THEN
	M_UserConfigure();
END_IF

//
// Set next state based on cfg.bAutoOp
//
IF cfg.bAutoOp THEN
	SetState(E_IODEV_STATE.OP, E_IODEV_SUBSTATE.OP_MONITORING);
ELSE
	// Monitoring but cannot activate outputs
	SetState(E_IODEV_STATE.NOTOP, E_IODEV_SUBSTATE.NOTOP_READY);
END_IF
END_METHOD

METHOD M_GetRpcErrorText : STRING
VAR_INPUT
	ErrorCode:	INT;
END_VAR
VAR
	str:	STRING;
END_VAR
CASE ErrorCode OF
	E_IODEV_RPC_ERROR.OK:						str	:= 'OK';
	E_IODEV_RPC_ERROR.NOT_OP:					str	:= 'Cannot control function. Not in OP state.';
	E_IODEV_RPC_ERROR.NOT_NOTOP_READY:		str	:= 'Call failed. Not in NOTOP/(READY or MONITORING).';
	E_IODEV_RPC_ERROR.NOT_NOTOP_NOTREADY:		str	:= 'Call failed. Not in NOTOP_NOTREADY/ERROR.';
	E_IODEV_RPC_ERROR.LOCAL:					str	:= 'RPC calls not allowed in Local mode.';
ELSE
	str	:= 'Unregistered RPC error.';
END_CASE

M_GetRpcErrorText	:= str;
END_METHOD

METHOD M_LogEventDebug : BOOL
VAR_INPUT
	sText:	STRING	:= '';
END_VAR
// Log Debug events only if both logging and debugging is enabled
IF  cfg.bLog AND cfg.bDebug THEN
	fbEventDebug.ipArguments.Clear().AddString(sText);
	fbEventDebug.Send(0);
END_IF
END_METHOD

METHOD M_LogEventError : BOOL
VAR_INPUT
	sText:	STRING	:= '';
END_VAR
// Log only if logging is enabled
IF  NOT cfg.bLog THEN
	RETURN;
END_IF

fbEventError.ipArguments.Clear().AddString(sText);
fbEventError.Send(0);
END_METHOD

METHOD M_LogEventGeneral : BOOL
VAR_INPUT
	sText:	STRING	:= '';
END_VAR
// Log only if logging is enabled
IF  NOT cfg.bLog THEN
	RETURN;
END_IF

fbEventGeneral.ipArguments.Clear().AddString(sText);
fbEventGeneral.Send(0);
END_METHOD

METHOD M_ReadSensors
VAR_INPUT
END_VAR
VAR
	i:	int;
END_VAR
//
// Digital inputs are mapped to physical input signals.
// Assign preconfigured label depending on the value
//
IF pArrDI <> 0 AND cfg.nNum_DI > 0  THEN
	FOR i := 0 TO (cfg.nNum_DI - 1) DO
		pArrDI[i].M_Compute();
	END_FOR
END_IF

//
// Analog inputs of type INT are mapped to physical input signals.
// Compute the reading in User Units
//
IF pArrAI <> 0 AND cfg.nNum_AI > 0  THEN
	FOR i := 0 TO (cfg.nNum_AI - 1) DO
		pArrAI[i].M_Compute();
	END_FOR
END_IF

//
// Analog inputs of type REAL are mapped to physical input signals.
// Compute the reading in User Units
//
IF pArrRI <> 0 AND cfg.nNum_RI > 0  THEN
	FOR i := 0 TO (cfg.nNum_RI - 1) DO
		pArrRI[i].M_Compute();
	END_FOR
END_IF
END_METHOD

METHOD M_ResetConfig
VAR_INPUT
END_VAR
VAR
	i:	int;
END_VAR
//
// Reset Digital inputs.
//
IF pArrDI <> 0 AND cfg.nNum_DI > 0  THEN
	FOR i := 0 TO (cfg.nNum_DI - 1) DO
		pArrDI[i].M_Reset();
	END_FOR
END_IF

//
// Reset Digital outputs.
//
IF pArrDO <> 0 AND cfg.nNum_DO > 0  THEN
	FOR i := 0 TO (cfg.nNum_DO - 1) DO
		pArrDO[i].M_Reset();
	END_FOR
END_IF

//
// Reset Analog inputs of type INT
//
IF pArrAI <> 0 AND cfg.nNum_AI > 0  THEN
	FOR i := 0 TO (cfg.nNum_AI - 1) DO
		pArrAI[i].M_Reset();
	END_FOR
END_IF

//
// Reset Analog inputs of type REAL
//
IF pArrRI <> 0 AND cfg.nNum_RI > 0  THEN
	FOR i := 0 TO (cfg.nNum_RI - 1) DO
		pArrRI[i].M_Reset();
	END_FOR
END_IF

//
// Reset Analog outputs.
//
IF pArrAO <> 0 AND cfg.nNum_AO > 0  THEN
	FOR i := 0 TO (cfg.nNum_AO - 1) DO
		pArrAO[i].M_Reset();
	END_FOR
END_IF
END_METHOD

METHOD M_ResetOutputs
VAR_INPUT
END_VAR
VAR
	i:	int;
END_VAR
//
// Reset digital outputs.
//
IF pArrDO <> 0 AND cfg.nNum_DO > 0  THEN
	FOR i := 0 TO (cfg.nNum_DO - 1) DO
		pArrDO[i].M_Reset();
	END_FOR
END_IF

//
// Reset analog outputs.
//
IF pArrAO <> 0 AND cfg.nNum_AO > 0  THEN
	FOR i := 0 TO (cfg.nNum_AO - 1) DO
		pArrAO[i].M_Reset();
	END_FOR
END_IF
END_METHOD

METHOD M_SetOutputs
VAR_INPUT
END_VAR
VAR
	i:	int;
END_VAR
//
// Set digital outputs.
//
IF pArrDO <> 0 AND cfg.nNum_DO > 0  THEN
	FOR i := 0 TO (cfg.nNum_DO - 1) DO
		pArrDO[i].M_Compute();
	END_FOR
END_IF

//
// Set analog outputs.
//
IF pArrAO <> 0 AND cfg.nNum_AO > 0  THEN
	FOR i := 0 TO (cfg.nNum_AO - 1) DO
		pArrAO[i].M_Compute();
	END_FOR
END_IF
END_METHOD

METHOD M_SetRpcStatus : INT
VAR_INPUT
	nErrorCode:	E_IODEV_RPC_ERROR;
END_VAR
RefStat.nRpcErrorCode	:= nErrorCode;
RefStat.sRpcErrorText	:= M_GetRpcErrorText(nErrorCode);

M_SetRpcStatus		:= nErrorCode;
END_METHOD

METHOD M_UserConfigure
VAR_INPUT
END_VAR
END_METHOD

METHOD ProcessEvents
VAR_INPUT
END_VAR

(* 
	Before processing the event, execute the Do-Activity tasks. 
	Note that, in case of orthogonal regions, more than one Do-Activity 
	could run in the same PLC cycle.
	Note: Most of these activities have timeouts since they take time.
*)

IF	RefStat.nSubstate = E_IODEV_SUBSTATE.OP_MONITORING OR 
	RefStat.nSubstate = E_IODEV_SUBSTATE.NOTOP_READY	THEN
	ActivityMonitoring();
END_IF



(* 
	Evaluate state machine transitions.
*)

CASE RefStat.nState OF

//***********************************
// NOTOP
//***********************************
E_IODEV_STATE.NOTOP:

	(* Transitions from NOTOP substates *)
	CASE RefStat.nSubstate OF
	
	E_IODEV_SUBSTATE.NOTOP_NOTREADY:		
		IF nEvent = E_IODEV_EVENT.INIT THEN
			ActionInitExecute();
			// Set next state based on cfg.bAutoOp
			IF cfg.bAutoOp THEN
				// Go directly to operational
				M_LogEventGeneral('Going to OP_MONITORING state.');
				SetState(E_IODEV_STATE.OP, E_IODEV_SUBSTATE.OP_MONITORING);
			ELSE
				// Monitoring but cannot activate outputs
				M_LogEventGeneral('Going to NOTOP_READYstate.');
				SetState(E_IODEV_STATE.NOTOP, E_IODEV_SUBSTATE.NOTOP_READY);
			END_IF
			RETURN;
		END_IF
		
	E_IODEV_SUBSTATE.NOTOP_READY:			
		IF nEvent = E_IODEV_EVENT.ENABLE THEN
			M_LogEventGeneral('ENABLE executed.');
			SetState(E_IODEV_STATE.OP, E_IODEV_SUBSTATE.OP_MONITORING);
			RETURN;
		END_IF

	E_IODEV_SUBSTATE.NOTOP_ERROR:			
		IF nEvent = E_IODEV_EVENT.HWOK THEN
			M_LogEventGeneral('Recovered from ERROR.');
			SetState(E_IODEV_STATE.NOTOP, E_IODEV_SUBSTATE.NOTOP_NOTREADY);
			RETURN;
		END_IF
		
	END_CASE

	(* Transitions from NOTOP state *)
	IF nEvent = E_IODEV_EVENT.ERRHW THEN
		ActionUnexpExecute();
		SetState(E_IODEV_STATE.NOTOP, E_IODEV_SUBSTATE.NOTOP_ERROR);
		RETURN;
	END_IF
	
//***********************************
// OPERATIONAL
//***********************************
E_IODEV_STATE.OP:

	(* Transitions from OP subastates *)
	CASE RefStat.nSubstate OF
	E_IODEV_SUBSTATE.OP_ERROR:			
		IF nEvent = E_IODEV_EVENT.HWOK THEN
			M_LogEventGeneral('Recovered from ERROR.');
			SetStatus(E_IODEV_ERROR.OK, 'OK');
			SetState(E_IODEV_STATE.OP, E_IODEV_SUBSTATE.OP_MONITORING);
			RETURN;			
		ELSIF nEvent = E_IODEV_EVENT.DISABLE THEN
			ActionDisableExecute();
			SetState(E_IODEV_STATE.NOTOP, E_IODEV_SUBSTATE.NOTOP_READY);
			RETURN;			
		END_IF

	E_IODEV_SUBSTATE.OP_MONITORING:			
		IF nEvent = E_IODEV_EVENT.SET THEN
			ActionSetExecute();
			RETURN;
		ELSIF nEvent = E_IODEV_EVENT.DISABLE THEN
			ActionDisableExecute();
			SetState(E_IODEV_STATE.NOTOP, E_IODEV_SUBSTATE.NOTOP_READY);
			RETURN;			
		END_IF
		
	END_CASE
	
	// Transitions from OP state.
	// Valid for any OP substate.
	IF nEvent = E_IODEV_EVENT.ERRHW THEN
		ActionUnexpExecute();
		SetState(E_IODEV_STATE.OP, E_IODEV_SUBSTATE.OP_ERROR);
		RETURN;
	END_IF
	
END_CASE

(* 
	"Global" internal transitions valid in any state should go here.
	They do not change the active state configuration. 
	They are evaluated after all the others transitions have been 
	considered.
*) 
IF nEvent = E_IODEV_EVENT.RESET THEN
	ActionResetExecute();
	SetState(E_IODEV_STATE.NOTOP, E_IODEV_SUBSTATE.NOTOP_NOTREADY);
	RETURN;
ELSIF
	nEvent = E_IODEV_EVENT.STOP THEN
	ActionStopExecute();
	RETURN;
END_IF
END_METHOD

{attribute 'TcRpcEnable':='1'}
METHOD RPC_Disable : INT
VAR_INPUT
END_VAR
// RPC calls are not allowed in Local mode.
IF RefStat.bLocal THEN
	RPC_Disable	:= M_SetRpcStatus(E_IODEV_RPC_ERROR.LOCAL);
	RETURN;
END_IF

// Disable command is accepted only if device is in OP state.
IF RefStat.nState <> E_IODEV_STATE.OP THEN
	RPC_Disable	:= M_SetRpcStatus(E_IODEV_RPC_ERROR.NOT_OP);
	RETURN;
ELSE
	// Set disable command
	RefCtrl.nCommand := E_IODEV_COMMAND.DISABLE;
	RefCtrl.bExecute := TRUE;

	// Call was successful
	RPC_Disable	:= M_SetRpcStatus(E_IODEV_RPC_ERROR.OK);
END_IF
END_METHOD

{attribute 'TcRpcEnable':='1'}
METHOD RPC_Enable : INT
VAR_INPUT
END_VAR
// RPC calls are not allowed in Local mode.
IF RefStat.bLocal THEN
	RPC_Enable	:= M_SetRpcStatus(E_IODEV_RPC_ERROR.LOCAL);
	RETURN;
END_IF

// Enable command is accepted only if device is in NOTOP_READY.
// Enable command is ignored (in ProcessEvents) in OP_MONITORING.
IF	RefStat.nSubstate <> E_IODEV_SUBSTATE.NOTOP_READY	AND
	RefStat.nSubstate <> E_IODEV_SUBSTATE.OP_MONITORING	THEN
	RPC_Enable	:= M_SetRpcStatus(E_IODEV_RPC_ERROR.NOT_NOTOP_READY);
	RETURN;
ELSE
	// Set enable command
	RefCtrl.nCommand := E_IODEV_COMMAND.ENABLE;
	RefCtrl.bExecute := TRUE;
	
	// Call was successful
	RPC_Enable	:= M_SetRpcStatus(E_IODEV_RPC_ERROR.OK);
END_IF
END_METHOD

{attribute 'TcRpcEnable':='1'}
METHOD RPC_Init : INT
VAR_INPUT
END_VAR
// RPC calls are not allowed in Local mode.
IF RefStat.bLocal THEN
	RPC_Init	:= M_SetRpcStatus(E_IODEV_RPC_ERROR.LOCAL);
	RETURN;
END_IF

// Init command is accepted only if device is in NOTOP_NOTREADY or ERROR.
IF 	RefStat.nSubstate <> E_IODEV_SUBSTATE.NOTOP_NOTREADY  AND  
	RefStat.nSubstate <> E_IODEV_SUBSTATE.NOTOP_ERROR 		THEN
	RPC_Init	:= M_SetRpcStatus(E_IODEV_RPC_ERROR.NOT_NOTOP_NOTREADY);
	RETURN;
ELSE
	// Set INIT command
	RefCtrl.nCommand := E_IODEV_COMMAND.INIT;
	RefCtrl.bExecute := TRUE;

	// Call was successful
	RPC_Init	:= M_SetRpcStatus(E_IODEV_RPC_ERROR.OK);
END_IF
END_METHOD

{attribute 'TcRpcEnable':='1'}
METHOD RPC_Reset : INT
VAR_INPUT
END_VAR
// RPC calls are not allowed in Local mode.
IF RefStat.bLocal THEN
	RPC_Reset	:= M_SetRpcStatus(E_IODEV_RPC_ERROR.LOCAL);
	RETURN;
END_IF

RefCtrl.nCommand := E_IODEV_COMMAND.RESET;
RefCtrl.bExecute := TRUE;

// Call was successful
RPC_Reset	:= M_SetRpcStatus(E_IODEV_RPC_ERROR.OK);
END_METHOD

{attribute 'TcRpcEnable':='1'}
METHOD RPC_SetDebug : INT
VAR_INPUT
	in_bDebug:	BOOL 	:= FALSE;		// If TRUE, activate event logging of Debug type
END_VAR
// Enable/disable Debugging
cfg.bDebug	:= in_bDebug;

// Call was successful
RPC_SetDebug	:= M_SetRpcStatus(E_IODEV_RPC_ERROR.OK);
END_METHOD

{attribute 'TcRpcEnable':='1'}
METHOD RPC_SetLog : INT
VAR_INPUT
	in_bLog:	BOOL 	:= FALSE;		// If TRUE, activate event logging
END_VAR
// Enable/disable Logging
cfg.bLog	:= in_bLog;

// Call was successful
RPC_SetLog	:= M_SetRpcStatus(E_IODEV_RPC_ERROR.OK);
END_METHOD

{attribute 'TcRpcEnable':='1'}
METHOD RPC_SetOutputs : INT
VAR_INPUT
END_VAR
// RPC calls are not allowed in Local mode.
IF RefStat.bLocal THEN
	RPC_SetOutputs	:= M_SetRpcStatus(E_IODEV_RPC_ERROR.LOCAL);
	RETURN;
END_IF

// SET command is accepted only in OP state.
IF RefStat.nState <> E_IODEV_STATE.OP THEN
	RPC_SetOutputs	:= M_SetRpcStatus(E_IODEV_RPC_ERROR.NOT_OP);
	RETURN;
ELSE
	// Set SET command
	RefCtrl.nCommand := E_IODEV_COMMAND.SET_OUTPUTS;
	RefCtrl.bExecute := TRUE;
	
	// Call was successful
	RPC_SetOutputs	:= M_SetRpcStatus(E_IODEV_RPC_ERROR.OK);
END_IF
END_METHOD

{attribute 'TcRpcEnable':='1'}
METHOD RPC_Stop : INT
VAR_INPUT
END_VAR
// RPC calls are not allowed in Local mode.
IF RefStat.bLocal THEN
	RPC_Stop	:= M_SetRpcStatus(E_IODEV_RPC_ERROR.LOCAL);
	RETURN;
END_IF

RefCtrl.nCommand := E_IODEV_COMMAND.STOP;
RefCtrl.bExecute := TRUE;

// Call was successful
RPC_Stop	:= M_SetRpcStatus(E_IODEV_RPC_ERROR.OK);
END_METHOD

METHOD SetAction
VAR_INPUT
	actionName:		STRING;
END_VAR


RefStat.sActionDesc := actionName;
END_METHOD

METHOD SetEvent
VAR_INPUT
	nEventId:			DINT;
END_VAR

nEvent := nEventId;

CASE nEventId OF
	E_IODEV_EVENT.NONE:
		RefStat.sEventDesc := '';
		RETURN;
		
	E_IODEV_EVENT.RESET:
		RefStat.sEventDesc := 'CMD RESET';
		RETURN;
	
	E_IODEV_EVENT.INIT:
		RefStat.sEventDesc := 'CMD INIT';
		RETURN;

	E_IODEV_EVENT.STOP:
		RefStat.sEventDesc := 'CMD STOP';
		RETURN;

	E_IODEV_EVENT.ENABLE:
		RefStat.sEventDesc := 'CMD ENABLE';
		RETURN;

	E_IODEV_EVENT.DISABLE:
		RefStat.sEventDesc := 'CMD DISABLE';
		RETURN;

	(* events corresponding to internal events *)
	(* evetnts mapped to HW signals *)
	E_IODEV_EVENT.SET:
		RefStat.sEventDesc := 'CMD SET';
		RETURN;

	E_IODEV_EVENT.INITDONE:
		RefStat.sEventDesc := 'SIG INITDONE';
		RETURN;

	E_IODEV_EVENT.HWOK:
		RefStat.sEventDesc := 'SIG HWOK';
		RETURN;

	E_IODEV_EVENT.ERRHW:
		RefStat.sEventDesc := 'INT ERRHW';
		RETURN;

	E_IODEV_EVENT.ERRINIT:
		RefStat.sEventDesc := 'INT ERRINIT';
		RETURN;

	
END_CASE 

(* INTERNAL ERROR *)
RefStat.sEventDesc := 'UNKNOWN EVENT';
END_METHOD

METHOD SetLastCommand
VAR_INPUT
	cmd:	E_IODEV_COMMAND;
END_VAR
RefStat.nLastCommand	:= cmd;

CASE cmd OF
	E_IODEV_COMMAND.RESET:
		RefStat.sLastCommand	:= 'RESET';
	E_IODEV_COMMAND.INIT:
		RefStat.sLastCommand	:= 'INIT';
	E_IODEV_COMMAND.STOP:
		RefStat.sLastCommand	:= 'STOP';
	E_IODEV_COMMAND.ENABLE:
		RefStat.sLastCommand	:= 'ENABLE';
	E_IODEV_COMMAND.DISABLE:
		RefStat.sLastCommand	:= 'DISABLE';
	E_IODEV_COMMAND.SET_OUTPUTS:
		RefStat.sLastCommand	:= 'SET';
ELSE
		RefStat.sLastCommand	:= 'NONE';
END_CASE;
END_METHOD

METHOD SetState : BOOL
VAR_INPUT
	nState:			E_IODEV_STATE;
	nSubstate:		E_IODEV_SUBSTATE;
END_VAR
(* 
	Update State Machine active state configuration.

	ToDo: support initial pseudo state/substate.
*)

IF nState <> E_IODEV_STATE.NONE THEN
	RefStat.nState	:= nState;
END_IF
IF nSubstate <> E_IODEV_SUBSTATE.NONE THEN
	RefStat.nSubstate	:= nSubstate;
END_IF

(* Update active state configuration description *)

IF nState = E_IODEV_STATE.NOTOP THEN
	RefStat.sState	:= 'NOT OP';
ELSIF nState = E_IODEV_STATE.OP THEN
	RefStat.sState	:= 'OPERATIONAL';
END_IF

IF nSubstate = E_IODEV_SUBSTATE.NOTOP_NOTREADY THEN
	RefStat.sSubstate	:= 'NOT READY';
ELSIF nSubstate = E_IODEV_SUBSTATE.NOTOP_READY THEN
	RefStat.sSubstate	:= 'READY';
ELSIF nSubstate = E_IODEV_SUBSTATE.NOTOP_ERROR THEN
	RefStat.sSubstate	:= 'ERROR';
ELSIF nSubstate = E_IODEV_SUBSTATE.OP_MONITORING THEN
	RefStat.sSubstate	:= 'MONITORING';
ELSIF nSubstate = E_IODEV_SUBSTATE.OP_ERROR THEN
	RefStat.sSubstate	:= 'ERROR';
ELSE
	RefStat.sSubstate	:= '';
END_IF


SetState	:= TRUE;
END_METHOD

METHOD SetStatus
VAR_INPUT
	nErrorCode:	E_IODEV_ERROR;
	sErrorText:	STRING;
END_VAR
RefStat.nErrorCode 	:= nErrorCode;
RefStat.sErrorText 	:= sErrorText;

IF nErrorCode <> E_IODEV_ERROR.OK THEN
	RefStat.sStatus	:= 'ERROR';
	RefStat.nStatus	:= E_IODEV_STATUS.ERROR;
ELSE
	RefStat.sStatus	:= 'OK';
	RefStat.nStatus	:= E_IODEV_STATUS.OK;
END_IF
END_METHOD

END_FUNCTION_BLOCK

// POUs/Examples/FB_SENS_2_4A_2R_USER_CONFIG
// EXAMPLE: Customised FB_IODEV_BASE for 2 DI, 4 AI, 2 DO and 2 AO.
//          Overloaded M_UserConfigure() method for User Configuration of channels.
FUNCTION_BLOCK FB_SENS_2_4A_2R_USER_CONFIG EXTENDS FB_IODEV_BASE
VAR_INPUT
END_VAR
VAR_OUTPUT
END_VAR
VAR
	// Control parameters as in T_IODEV_CTRL
	{attribute 'OPC.UA.DA' := '1'}
	ctrl:	T_IODEV_CTRL;	
	// Status parameters that EXTEND T_IODEV_STAT
	{attribute 'OPC.UA.DA' := '1'}
	{attribute 'OPC.UA.DA.Access' := '1'}
	stat:	T_IODEV_STAT_2_4A_2R;	
END_VAR

//
// TODO_USER
//
//
// Set References
RefCtrl	REF=ctrl;
RefStat	REF=stat;

// Set number of channels for each type.
// Default values are set to zero.
// Set whatever is not zero, i.e. whatever is defined.
// WARNING: The values MUST match the sizes of corresponding arrays above !!!
//
cfg.nNum_DI		:=	2; 	// Number of digital INPUT signals,      arrDI:	ARRAY [0..1]
cfg.nNum_AI		:=	4; 	// Number of analog INT  INPUT signals,  arrAI:	ARRAY [0..3]
cfg.nNum_RI		:=	2; 	// Number of analog REAL INPUT signals,  arrRI:	ARRAY [0..3]


//
// Set pointers for EXISTING arrays ONLY, e.g. arrDI, arrAI, etc.
//
pArrDI	:= ADR(stat.arrDI[0]);
pArrAI	:= ADR(stat.arrAI[0]);
pArrRI	:= ADR(stat.arrRI[0]);

//
// Execute the base class object FB_IODEV_BASE
//
SUPER^();

// TODO_USER
//
// Define individual channel configurations, if used.
METHOD M_UserConfigure
VAR_INPUT
END_VAR
// TODO_USER
//
// Example implementation.
// Hard code any signal configuration.
//

// Configuration parameter cfg.bUserConfig defines if 
// the hard-coded configuration below should be used or
// the signals will be configured from the WS.

//
// Digital signals
//
// Digital inputs (defined in stat structure T_IODEV_STAT_CUSTOM)
// Signal DI[0] is a door open signal
// Signal DI[1] is a light switch signal
stat.arrDI[0].M_Configure('CLOSED', 'OPEN');
stat.arrDI[1].M_Configure('OFF',    'ON');


//
// Analog signals
//
// Analog inputs of type INT (defined in stat structure T_IODEV_STAT_2_4A_2R)
stat.arrAI[0].M_Configure(CONVERSION_IODEV_NONE, 		0.0,   0.0, 0.0);
stat.arrAI[1].M_Configure(CONVERSION_IODEV_LINEAR, 		2.0,   1.0, 0.0);
stat.arrAI[2].M_Configure(CONVERSION_IODEV_QUADRATIC,	2.0,   1.0, 5.0);
// Edwards pressure guage
// P =10^(1.5*V - 12)    [mbar]
// 16-bit A/D converter, +=10V, e.g. EL3102.
// 1V = 2^16/10/2 = 3276.8 bit
// P = 10^(1.5*V - 12) = 10^(1.5/3276.8*bit - 12) = 10^(0.000457763*bit - 12)
stat.arrAI[3].M_Configure(CONVERSION_IODEV_EXP10, 	0.000457763, -12.0, 0.0);	



//
// Analog inputs of type REAL (defined in stat structure T_IODEV_STAT_2_4A_2R)
//
stat.arrRI[0].M_Configure(CONVERSION_IODEV_NONE, 		0.0,   0.0, 0.0);
stat.arrRI[1].M_Configure(CONVERSION_IODEV_LINEAR, 		2.0,   1.0, 0.0);
END_METHOD

END_FUNCTION_BLOCK

// POUs/Examples/FB_SENS_8_4
// EXAMPLE: FB for SENSORS with 8 DI and 4 AI
FUNCTION_BLOCK FB_SENS_8_4 EXTENDS FB_IODEV_BASE
VAR_INPUT
END_VAR
VAR_OUTPUT
END_VAR
VAR
	// Control parameters as defined in T_IODEV_CTRL.
	// For sensors use the base control structure T_IODEV_CTRL.
	{attribute 'OPC.UA.DA' := '1'}
	ctrl:	T_IODEV_CTRL;	
	// Status parameters that EXTEND T_IODEV_STAT
	{attribute 'OPC.UA.DA' := '1'}
	{attribute 'OPC.UA.DA.Access' := '1'}
	stat:	T_IODEV_STAT_8_4;	
END_VAR

//
// TODO_USER
//
//
// Set References
RefCtrl	REF=ctrl;
RefStat	REF=stat;

// Set number of channels for each type.
// Default values are set to zero.
// Set whatever is not zero, i.e. whatever is defined.
// WARNING: The values MUST match the sizes of corresponding arrays above !!!
//
cfg.nNum_DI		:=	8; 	// Number of digital INPUT signals, arrDI:	ARRAY [0..7]
cfg.nNum_AI		:=	4; 	// Number of analog INPUT signals,  arrAI:	ARRAY [0..3]

//
// Set pointers for EXISTING arrays ONLY, e.g. arrDI, arrAI, etc.
//
pArrDI	:= ADR(stat.arrDI[0]);
pArrAI	:= ADR(stat.arrAI[0]);

//
// Execute the base class object FB_IODEV_BASE
//
SUPER^();

END_FUNCTION_BLOCK

// POUs/Examples/FB_SENS_8_4_USER_CONFIG
// EXAMPLE: Customised FB_SENS_8_4 with additional User Configuration of channels
//          Only the M_UserConfigure() method is added to FB_SENS_8_4.
FUNCTION_BLOCK FB_SENS_8_4_USER_CONFIG EXTENDS FB_SENS_8_4
VAR_INPUT
END_VAR
VAR_OUTPUT
END_VAR
VAR
END_VAR

//
// Execute the base class FB_IODEV_SENS_8_4 object.
//
SUPER^();

// TODO_USER
//
// Define individual channel configurations, if used.
METHOD M_UserConfigure
VAR_INPUT
END_VAR
// TODO_USER
//
// Example implementation.
// Hard code any signal configuration.
//

// Configuration parameter cfg.bUserConfig defines if 
// the hard-coded configuration below should be used or
// the signals will be configured from the WS.

//
// Digital inputs
// Signal DI[0] is a LASER ON/OFF signal
// Signal DI[1] is a motor RUNNING/STOPPED signal
stat.arrDI[0].M_Configure('LASER OFF', 'LASER ON');
stat.arrDI[1].M_Configure('MOTOR STOPPED', 'MOTOR RUNNING');


//
// Analog inputs
//
stat.arrAI[0].M_Configure(CONVERSION_IODEV_NONE, 		0.0,   0.0, 0.0);
stat.arrAI[1].M_Configure(CONVERSION_IODEV_LINEAR, 		2.0,   1.0, 0.0);
stat.arrAI[2].M_Configure(CONVERSION_IODEV_QUADRATIC,	2.0,   1.0, 5.0);
// Edwards pressure guage
// P =10^(1.5*V - 12)    [mbar]
// 16-bit A/D converter, +=10V, e.g. EL3102.
// 1V = 2^16/10/2 = 3276.8 bit
// P = 10^(1.5*V - 12) = 10^(1.5/3276.8*bit - 12) = 10^(0.000457763*bit - 12)
stat.arrAI[3].M_Configure(CONVERSION_IODEV_EXP10, 	0.000457763, -12.0, 0.0);
END_METHOD

END_FUNCTION_BLOCK

// POUs/Simulation/FB_SIM_SIGNAL_ANALOG
FUNCTION_BLOCK FB_SIM_SIGNAL_ANALOG
VAR_INPUT
	// q_nSignal = sin() * in_nScale + in_nOffset
	// in_nPeriod [ms] corresponds to 2PI angle
	in_nPeriod:	DINT	:= 10000;	// Period for signal to go o-max-0
	in_nScale:	LREAL 	:= 1.0;		// Scale of the output
	in_nOffset:	INT 	:= 0;		// Offset of the output
END_VAR
VAR_OUTPUT
END_VAR
VAR
	q_nSignal	AT %Q*:	INT;			//	Simulated output signal to be linked to analog sensor input
	
	timer:	TON;						// Timer ET and PT used for 'angle' for sin(). Angle = ET / PT * 2PI
	initialised:	BOOL := FALSE;		// Used to start timer for the first time
END_VAR
VAR_TEMP
	t1:	LREAL;
	t2:	LREAL;
	t3:	LREAL;
	t4:	LREAL;
END_VAR

IF NOT initialised THEN
	initialised := TRUE;
	
	// Start timer for signal=FALSE
	timer(IN:=FALSE);
	timer(IN:=TRUE, PT:=DINT_TO_TIME(in_nPeriod));
	RETURN;
END_IF

// Execute timer
// The timer is actually used just for the 'angle' for the sin().
// Angle = ET / PT * 2PI
timer();

// If the timer expired, just restart it
IF timer.Q THEN
		timer(IN:=FALSE);
		timer(IN:=TRUE, PT:=DINT_TO_TIME(in_nPeriod));
END_IF

// Set the output
t1	:= TIME_TO_LREAL(timer.ET);
t2	:= TIME_TO_LREAL(timer.PT);
t3	:= t1 / t2 * 2 * 3.14;
t4	:= in_nScale * SIN(t3);
q_nSignal := in_nOffset + LREAL_TO_INT(t4);

END_FUNCTION_BLOCK

// POUs/Simulation/FB_SIM_SIGNAL_DIGITAL
FUNCTION_BLOCK FB_SIM_SIGNAL_DIGITAL
VAR_INPUT
	in_nPeriodLow:	DINT	:= 10000;	// Period for signal = FALSE
	in_nPeriodHigh:	DINT	:= 1000;	// Period for signal = TRUE
END_VAR
VAR_OUTPUT
END_VAR
VAR
	q_bSignal	AT %Q*:	BOOL;			//	Simulated output signal to be linked to sensor input
	
	timer:	TON;
	initialised:	BOOL := FALSE;
END_VAR

IF NOT initialised THEN
	initialised := TRUE;
	
	// Set initial state of the simulated signal to FALSE
	q_bSignal := FALSE;
	
	// Start timer for signal=FALSE
	timer(IN:=FALSE);
	timer(IN:=TRUE, PT:=DINT_TO_TIME(in_nPeriodLow));
	RETURN;
END_IF

// Execute timer
timer();

// If the timer expired, swap the signal and start corresponding timer
IF timer.Q THEN
	IF q_bSignal = FALSE THEN
		q_bSignal := TRUE;
	
		// Start timer for signal=TRUE
		timer(IN:=FALSE);
		timer(IN:=TRUE, PT:=DINT_TO_TIME(in_nPeriodHigh));
	ELSE
		q_bSignal := FALSE;
	
		// Start timer for signal=FALSE
		timer(IN:=FALSE);
		timer(IN:=TRUE, PT:=DINT_TO_TIME(in_nPeriodLow));
	END_IF
END_IF

END_FUNCTION_BLOCK

// POUs/Simulation/FB_SIM_SIGNAL_REAL
FUNCTION_BLOCK FB_SIM_SIGNAL_REAL
VAR_INPUT
	// q_nSignal = sin() * in_nScale + in_nOffset
	// in_nPeriod [ms] corresponds to 2PI angle
	in_nPeriod:	DINT	:= 10000;	// Period [ms] for signal to go 0-max-0
	in_nScale:	LREAL 	:= 1.0;		// Scale of the output
	in_nOffset:	LREAL 	:= 0;		// Offset of the output
END_VAR
VAR_OUTPUT
END_VAR
VAR
	q_rSignal	AT %Q*:	REAL;			//	Simulated output signal to be linked to analog sensor input of type REAL
	
	timer:			TON;				// Timer ET and PT used for 'angle' for sin(). Angle = ET / PT * 2PI
	initialised:	BOOL := FALSE;		// Used to start timer for the first time
END_VAR
VAR_TEMP
	t1:	LREAL;
	t2:	LREAL;
	t3:	LREAL;
	t4:	LREAL;
END_VAR

IF NOT initialised THEN
	initialised := TRUE;
	
	// Start timer for signal=FALSE
	timer(IN:=FALSE);
	timer(IN:=TRUE, PT:=DINT_TO_TIME(in_nPeriod));
	RETURN;
END_IF

// Execute timer
// The timer is actually used just for the 'angle' for the sin().
// Angle = ET / PT * 2PI
timer();

// If the timer expired, just restart it
IF timer.Q THEN
		timer(IN:=FALSE);
		timer(IN:=TRUE, PT:=DINT_TO_TIME(in_nPeriod));
END_IF

// Set the output
t1	:= TIME_TO_LREAL(timer.ET);
t2	:= TIME_TO_LREAL(timer.PT);
t3	:= t1 / t2 * 2 * 3.14;
t4	:= in_nScale * SIN(t3);
q_rSignal := LREAL_TO_REAL(in_nOffset + t4);

END_FUNCTION_BLOCK

// POUs/MAIN
PROGRAM MAIN
VAR
sVer:	STRING := stLibVersion_ESO_LDC_IODev_Library.sVersion;

	// IMPORTANT:	In order to access RPC Calls via OPC UA, 
	//				attribute 'OPC.UA.DA':='1' is needed!!!
	{attribute 'OPC.UA.DA':='1'}
	IODev001:		FB_IODEV_2_4_2_2_USER_CONFIG;
	{attribute 'OPC.UA.DA':='1'}
	IODev002:		FB_SENS_8_4;
	{attribute 'OPC.UA.DA':='1'}
	IODev003:		FB_SENS_8_4_USER_CONFIG;
	{attribute 'OPC.UA.DA':='1'}
	IODev004:		FB_SENS_2_4A_2R_USER_CONFIG;
	
	// Simulated signals
	//
	// Digital
	SIM_bDig1:	FB_SIM_SIGNAL_DIGITAL;
	SIM_bDig2:	FB_SIM_SIGNAL_DIGITAL;
	
	// Analog
	SIM_nAnlg1:	FB_SIM_SIGNAL_ANALOG;
	SIM_nAnlg2:	FB_SIM_SIGNAL_ANALOG;
	SIM_nAnlg3:	FB_SIM_SIGNAL_ANALOG;
	SIM_nAnlg4:	FB_SIM_SIGNAL_ANALOG;

	SIM_rAnlg1:	FB_SIM_SIGNAL_REAL;
	SIM_rAnlg2:	FB_SIM_SIGNAL_REAL;
	
	q_nCouplerState	AT %Q*:	UINT := 8;	// Coupler state for full simulation

END_VAR

//
// Simulated signals
//
SIM_bDig1(in_nPeriodLow:=5000, in_nPeriodHigh:=2000);
SIM_bDig2(in_nPeriodLow:=2000, in_nPeriodHigh:=4000);

SIM_nAnlg1(in_nPeriod:=10000, in_nScale:=10000.0,	in_nOffset:=0);
SIM_nAnlg2(in_nPeriod:=10000, in_nScale:=100.0, 	in_nOffset:=5000);
SIM_nAnlg3(in_nPeriod:=10000, in_nScale:=10.0, 		in_nOffset:=1000);

// Simulation of Edwards pressure guage
// Vary input from 4.5 to 5.0 V 
// 16-bit A/D converter, +=10V, e.g. EL3102.
// 1V = 2^16/10/2 = 3276.8 bit
// 4.5 to 5.0 V ==> 4.5*3276.8 to 5.0*3276.8 bit ==> 14745 to 16384
// in_nScale = (16384 - 14745) / 2 = 819.5
// in_nOffset = 14745 + 819.5 = 15564.5
SIM_nAnlg4(in_nPeriod:=30000, in_nScale:=819.5, 	in_nOffset:=15564);


SIM_rAnlg1(in_nPeriod:=20000, in_nScale:=1000.0,	in_nOffset:=1000.0);
SIM_rAnlg2(in_nPeriod:=10000, in_nScale:=100.0,		in_nOffset:=0.0);


//
// Real devices
//

//
// IODev1
//
// The device will go directly to OP/MONITORING on PLC reboot.
// The configuration defined in M_UserConfigure() will be applied.
IODev001(	in_sName:='IODev001', in_bAutoOp:= TRUE, in_bUserConfig:=TRUE);

//
// IODev2
//
// The device will go directly to OP/MONITORING on PLC reboot.
// The configuration defined in M_UserConfigure() will NOT be applied.
IODev002(	in_sName:='IODev002', in_bAutoOp:= TRUE);
		
//
// IODev3
//
// The device will go directly to OP/MONITORING on PLC reboot.
// The configuration defined in M_UserConfigure() will be applied.
IODev003(	in_sName:='IODev003', in_bAutoOp:= TRUE, in_bUserConfig:=TRUE);

//
// IODev4
//
// The device will go directly to OP/MONITORING on PLC reboot.
// The configuration defined in M_UserConfigure() will be applied.
IODev004(	in_sName:='IODev004', in_bAutoOp:= TRUE, in_bUserConfig:=TRUE);

END_PROGRAM

// VISUs/Templates/GUI_TEMPLATE_IODEV
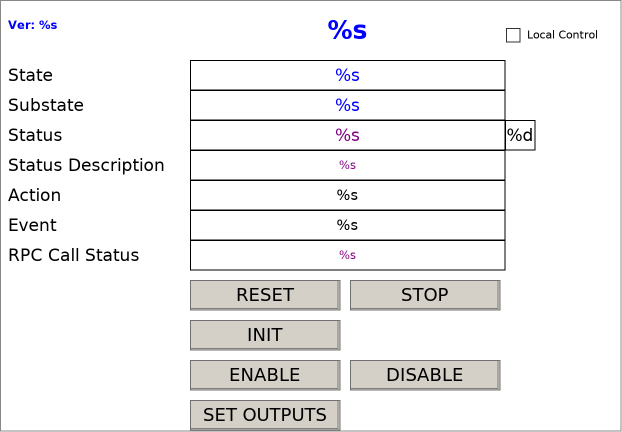
VISUALIZATION GUI_TEMPLATE_IODEV  // 622x432
VAR_IN_OUT
	m_Instance:	FB_IODEV_BASE;
END_VAR
    Rectangle (190,60 315x30), "%s", text variable: m_Instance.stat.sState
    Rectangle (190,90 315x30), "%s", text variable: m_Instance.stat.sSubstate
    Button (190,280 150x30), "RESET", input disabled if: (m_Instance.stat.bLocal = FALSE) <> 0
        OnMouseDown: execute { m_Instance.ctrl.nCommand := E_IODEV_COMMAND.RESET; m_Instance.ctrl.bExecute := TRUE; }
    Button (190,320 150x30), "INIT", input disabled if: (m_Instance.stat.bLocal = FALSE) <> 0
        OnMouseDown: execute { m_Instance.ctrl.nCommand := E_IODEV_COMMAND.INIT; m_Instance.ctrl.bExecute := TRUE; }
    Button (350,280 150x30), "STOP", input disabled if: (m_Instance.stat.bLocal = FALSE) <> 0
        OnMouseDown: execute { m_Instance.ctrl.nCommand := E_IODEV_COMMAND.STOP; m_Instance.ctrl.bExecute := TRUE; }
    Button (190,360 150x30), "ENABLE", input disabled if: (m_Instance.stat.bLocal = FALSE) <> 0
        OnMouseDown: execute { m_Instance.ctrl.nCommand := E_IODEV_COMMAND.ENABLE; m_Instance.ctrl.bExecute := TRUE; }
    Button (350,360 150x30), "DISABLE", input disabled if: (m_Instance.stat.bLocal = FALSE) <> 0
        OnMouseDown: execute { m_Instance.ctrl.nCommand := E_IODEV_COMMAND.DISABLE; m_Instance.ctrl.bExecute := TRUE; }
    Button (190,400 150x30), "SET OUTPUTS", input disabled if: (m_Instance.stat.bLocal = FALSE) <> 0
        OnMouseClick: execute { m_Instance.ctrl.nCommand := E_IODEV_COMMAND.SET_OUTPUTS; m_Instance.ctrl.bExecute := TRUE; }
    Rectangle (5,60 180x30), "State"
    Rectangle (5,90 180x30), "Substate"
    Rectangle (190,120 315x30), "%s", text variable: m_Instance.stat.sStatus
    Rectangle (190,150 315x30), "%s", text variable: m_Instance.stat.sErrorText
    Rectangle (5,120 180x30), "Status"
    Rectangle (5,150 180x30), "Status Description"
    Rectangle (190,180 315x30), "%s", text variable: m_Instance.stat.sActionDesc
    Rectangle (190,210 315x30), "%s", text variable: m_Instance.stat.sEventDesc
    Rectangle (5,180 180x30), "Action"
    Rectangle (5,210 180x30), "Event"
    Rectangle (190,12 315x35), "%s", text variable: m_Instance.cfg.sName
    Rectangle (505,120 30x30), "%d", text variable: m_Instance.stat.nStatus
    Checkbox (504,20 116x30), "Local Control", variable: m_Instance.stat.bLocal
    Rectangle (190,240 315x30), "%s", text variable: m_Instance.stat.sRPCErrorText
    Rectangle (5,240 180x30), "RPC Call Status"
    Rectangle (5,10 99x30), "Ver: %s", tooltip "'IODev.library version'", text variable: m_Instance.stat.sLibVersion, input disabled if: true
END_VISUALIZATION

// VISUs/GUI_IODev001
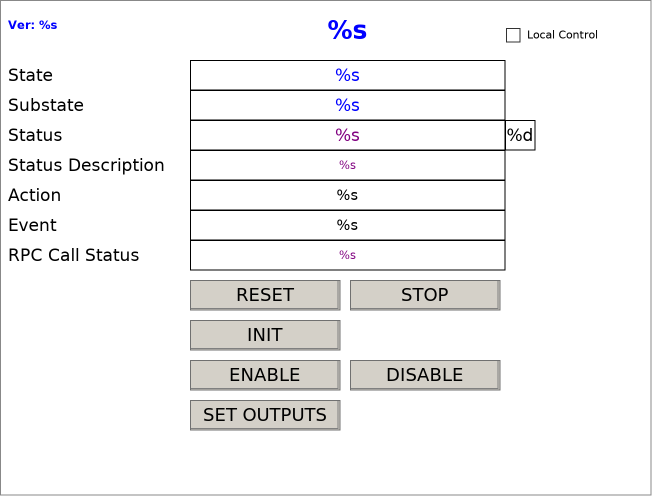
VISUALIZATION GUI_IODev001  // 652x496
    Frame (0,0 650x494)
        shows GUI_TEMPLATE_IODEV(m_Instance := MAIN.IODev001)
END_VISUALIZATION

// VISUs/GUI_IODev002
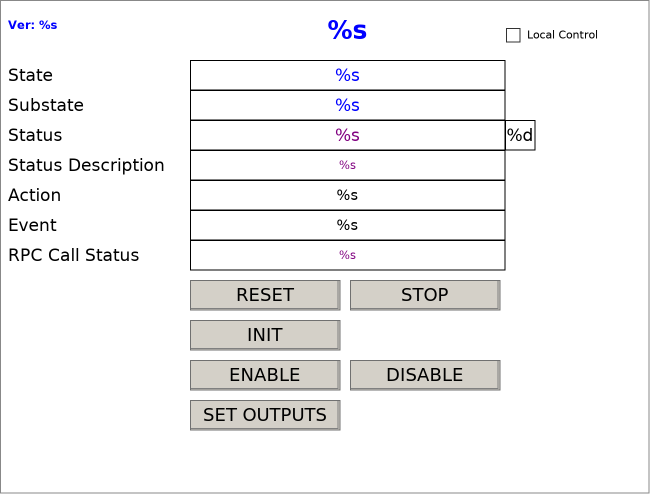
VISUALIZATION GUI_IODev002  // 650x494
    Frame (0,0 650x494)
        shows GUI_TEMPLATE_IODEV(m_Instance := MAIN.IODev002)
END_VISUALIZATION
